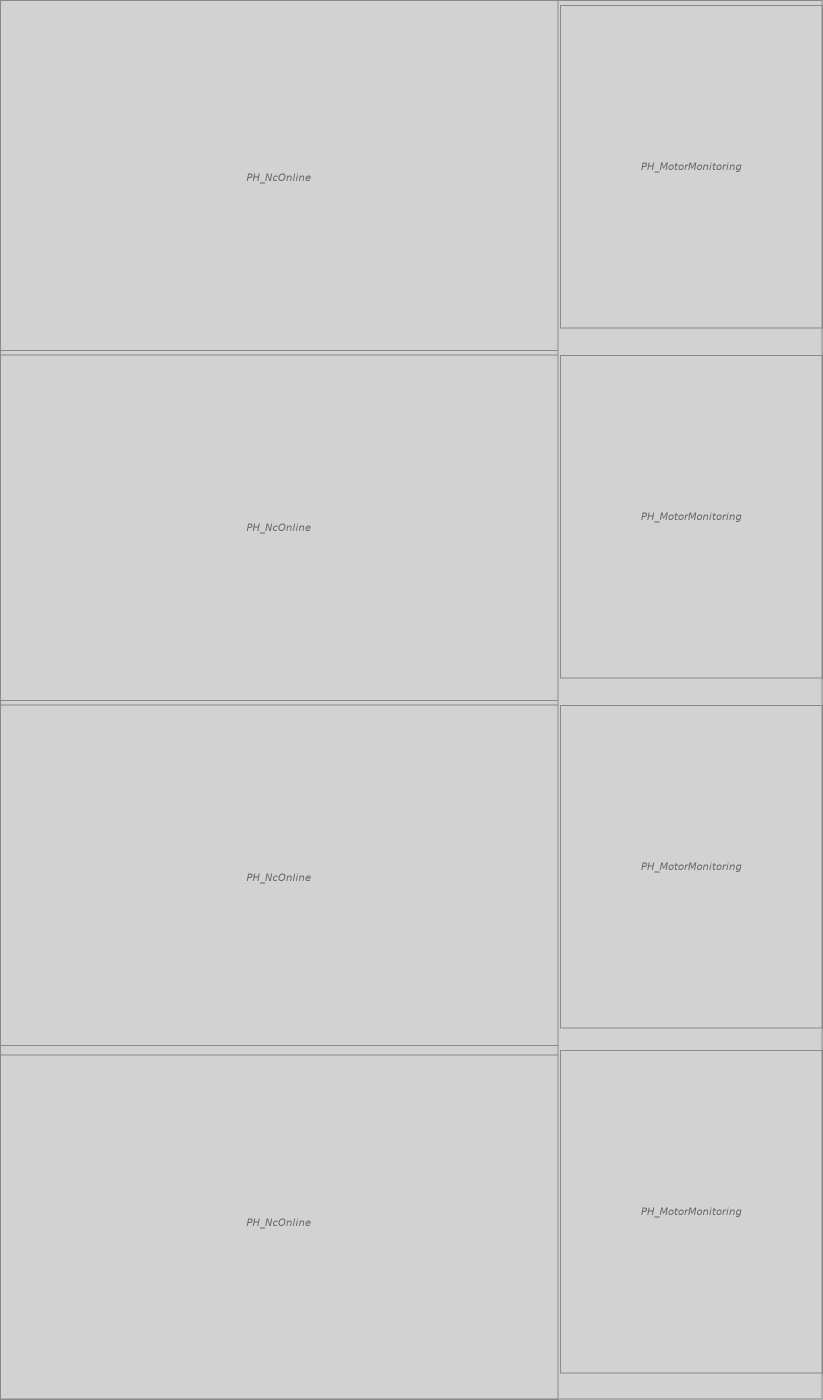
VISUALIZATION V_MainVisu  // 823x1400
    Frame (0,0 558x355)
        shows PH_NcOnline(stMcAxisOnline := GVL.aAxis[1])
    Frame (0,350 558x355)
        shows PH_NcOnline(stMcAxisOnline := GVL.aAxis[2])
    Frame (0,700 558x355)
        shows PH_NcOnline(stMcAxisOnline := GVL.aAxis[3])
    Frame (560,705 263x323)
        shows PH_MotorMonitoring(stMcAxisOnline := GVL.aAxis[3])
    Frame (560,355 263x323)
        shows PH_MotorMonitoring(stMcAxisOnline := GVL.aAxis[2])
    Frame (560,5 263x323)
        shows PH_MotorMonitoring(stMcAxisOnline := GVL.aAxis[1])
    Frame (0,1045 558x355)
        shows PH_NcOnline(stMcAxisOnline := GVL.aAxis[4])
    Frame (560,1050 263x323)
        shows PH_MotorMonitoring(stMcAxisOnline := GVL.aAxis[4])
END_VISUALIZATION

(* stored: Version 1.1.0.1, ProductVersion 3.1.4026.12
   Visu V_MainVisu: Id {82432f4a-f7cb-4c59-9a7d-462b886de51d} *)
